Yaskawa INFORM job: KAMERA.JBI

/JOB
//NAME KAMERA
///FOLDERNAME INNE
//POS
///NPOS 10,10,0,0,0,0
///TOOL 0
///POSTYPE PULSE
///PULSE
C00000=40550,-49639,-20907,0,63857,1
C00001=109961,-49639,-20907,0,63857,1
C00002=169926,-49639,-20907,0,63857,1
C00003=150403,-17087,28621,39932,45195,-16047
C00004=156447,-12587,35560,42339,37169,-16791
C00005=156447,-12587,35560,42339,37169,-16791
C00006=140702,2292,67612,56432,36179,-28502
C00007=133320,-12979,45062,50308,43228,-26962
C00008=109961,-49639,-20907,0,63857,1
C00009=40550,-49639,-20907,0,63857,1
BC00000=370339,142528,820160
BC00001=368238,63310,820163
BC00002=368238,13758,820163
BC00003=368238,13758,820160
BC00004=368238,13758,820160
BC00005=368238,13758,820160
BC00006=368238,13758,820160
BC00007=368238,13758,820160
BC00008=368238,63310,820163
BC00009=370339,142528,820160
//INST
///DATE 2023/11/01 18:40
///ATTR SC,RW
///GROUP1 RB1,BS1
NOP
MOVJ C00000 BC00000 VJ=50.00
MOVJ C00001 BC00001 VJ=50.00
MOVJ C00002 BC00002 VJ=50.00
MOVJ C00003 BC00003 VJ=50.00
MOVL C00004 BC00004 V=83.3
MOVL C00005 BC00005 V=83.3 PL=0
MACRO1 MJ#(0) ARGF10
ARCON
MOVL C00006 BC00006 V=13.3
ARCOF
MOVL C00007 BC00007 V=83.3
MOVJ C00008 BC00008 VJ=50.00
MOVJ C00009 BC00009 VJ=50.00
END
